                                                                       //
	//Sprawdzanie platynek                                              //
	bLidPuttedCheckEnableShow      						: BOOL;  		//	P030_Recipes.stActRecipe.stUBL.bLidPuttedCheckEnableShow   			// Zezwolenie na prace stacji sprawdzania nakrętek
    lrLidPuttedCheckHeightSVShow 	 					: LREAL;        //    P030_Recipes.stActRecipe.stUBL.lrLidPuttedCheckHeightSVShow			
	lrLidPuttedCheckPositionShow						: LREAL;		//	P030_Recipes.stActRecipe.stUBL.lrLidPuttedCheckPositionShow			// Pozycka sprawdzania platynki
	lrLidPuttedCheckAreaShow							: LREAL;		//	P030_Recipes.stActRecipe.stUBL.lrLidPuttedCheckAreaShow				// [-50...50]  lrLidPuttedCheckPosition +- lrLidPuttedCheckArea. Granica monitorowania 
	iLidPuttedCheckProgramShow							: INT;			//	P030_Recipes.stActRecipe.stUBL.iLidPuttedCheckProgramShow				// Program czujnika wizyjnego 0-20
                                                                        //
	//Zgrzewanie                                                        //
	bLidSealerEnableShow								: BOOL;			//	P030_Recipes.stActRecipe.stUBL.bLidSealerEnableShow				// Zezwolenie na pracę podajnika 
    bLidSealerHeaterEnableShow							: BOOL;			//	P030_Recipes.stActRecipe.stUBL.bLidSealerHeaterEnableShow			// Zezwolenie na prace grzałki  
    iLidSealerHeatingTimeShow							: INT;			//	P030_Recipes.stActRecipe.stUBL.iLidSealerHeatingTimeShow			// Czas zgrzewania  [ms]
	lrLidSealerPressureShow								: LREAL;		//	P030_Recipes.stActRecipe.stUBL.lrLidSealerPressureShow				//	Siła zgrzewania [kg] 
  	lrLidSealerHeightPosSVShow							: LREAL;		//	P030_Recipes.stActRecipe.stUBL.lrLidSealerHeightPosSVShow			// Wysokoć na której ma znajdować się grzałka
	iLidSealerTempHisteresisShow						: INT;			//	P030_Recipes.stActRecipe.stUBL.iLidSealerTempHisteresisShow		// Histereza poprawnej temperatury grzałki (+/- *C), po jej przekroczeniu grzałka wpada w błšd
   	iLidSealer1TempSVShow								: INT;			//	P030_Recipes.stActRecipe.stUBL.iLidSealer1TempSVShow				// Temperatura zadana grzałki 1                                                               
  	iLidSealer2TempSVShow								: INT;			//	P030_Recipes.stActRecipe.stUBL.iLidSealer2TempSVShow				// Temperatura zadana grzałki 2
                                                                        //
	//Przeciąganie zgrzewania                                           //
	bLidSealerDragingStationEnableShow					: BOOL;			//	P030_Recipes.stActRecipe.stUBL.bLidSealerDragingStationEnableShow					// Aktywacja przeciagania formatek pod zakrecarkami
	lrLidSealerDragingStationVelocityShow				: LREAL; 		//	P030_Recipes.stActRecipe.stUBL.lrLidSealerDragingStationVelocityShow				// Prędkosć przeciągania formatek pod zakręcarkami [0-100 %]
    lrLidSealerDragingStationAccelerationShow			: LREAL; 		//	P030_Recipes.stActRecipe.stUBL.lrLidSealerDragingStationAccelerationShow		// Przyspieszenie przeciągania formatek pod podajnikem płatynek 	
    lrLidSealerDragingStationDecelerationShow			: LREAL; 		//	P030_Recipes.stActRecipe.stUBL.lrLidSealerDragingStationDecelerationShow		// Zmniejszenie prędkości przeciągania formatek pod podajnikem płatynek 	
                                                                        //
	//Szlaban podawania zamknięć                            			//	
	bCapFeederGateEnableShow							:BOOL;			//	P030_Recipes.stActRecipe.stUBL.bCapFeederGateEnableShow				// Aktywacja 
	iCapFeederGateBlockingTimeShow						:INT;			//	P030_Recipes.stActRecipe.stUBL.iCapFeederGateBlockingTimeShow		// Czas blokowania
                                                                        //
	//[H] Podajnik zamknięć                        				        //
	bCapFeederEnableShow								:BOOL;			//	P030_Recipes.stActRecipe.stUBL.bCapFeederEnableShow							// [H] Aktywacja
    lrCapFeederHeightPosSVShow							:LREAL:=140;	//	P030_Recipes.stActRecipe.stUBL.lrCapFeederHeightPosSVShow						// [H] Pozycja
	iCapFeederTimeDelayOnShow							:INT; 			//	P030_Recipes.stActRecipe.stUBL.iCapFeederTimeDelayOnShow						// [H] Opóźnienie włączenia
	iCapFeederTimeDelayOffShow							:INT; 			//	P030_Recipes.stActRecipe.stUBL.iCapFeederTimeDelayOffShow						// [H] Opóźnienie wyłączenia
	iCapFeederTimeToEmptySleeveErrorShow				:INT;			//	P030_Recipes.stActRecipe.stUBL.iCapFeederTimeToEmptySleeveErrorShow			// [H] Czas do alarmu pustego rękawa [s] (10-120 s)
                                                                        //
	//Sorter nasadek                                                    //
	//Zmienne z innego sterownika                                       //
	bCapSorterOnlyWeightOKEnableShow					:BOOL;			//	P030_Recipes.stActRecipe.stUBL.bCapSorterOnlyWeightOKEnableShow		// Nakładanie zamknięć tylko na opakowania z waga OK
	                                                                    //
	//Przeciąganie pod sorterem nasadek                                 //
	bCapSorterDragEnableShow							:BOOL;			//	P030_Recipes.stActRecipe.stUBL.bCapSorterDragEnableShow				// [H] Aktywacja
	lrCapSorterDragVelocityShow							:LREAL; 		//	P030_Recipes.stActRecipe.stUBL.lrCapSorterDragVelocityShow				// Prędkość
 	lrCapSorterDragAccelerationShow						:LREAL;			//	P030_Recipes.stActRecipe.stUBL.lrCapSorterDragAccelerationShow			// Przyspieszenie 
	lrCapSorterDragDecelerationShow						:LREAL;			//	P030_Recipes.stActRecipe.stUBL.lrCapSorterDragDecelerationShow			// Hamowanie
                                 				                        //
	//Sprawdzanie nasadki                                      			//	
	bCapPuttedCheckEnableShow							:BOOL;			//	P030_Recipes.stActRecipe.stUBL.bCapPuttedCheckEnableShow				// Aktywacja
    lrCapPuttedCheckHeightPosSVShow						:LREAL:=69;		//	P030_Recipes.stActRecipe.stUBL.lrCapPuttedCheckHeightPosSVShow			// Pozycja
                                 					                    //
	//Zakrecarka szczekowa (Zachować kolejność i opisy!)                //
	bGripperScrewer1EnableShow							:BOOL;			//	P030_Recipes.stActRecipe.stUBL.bGripperScrewer1EnableShow								// Aktywacja 1
	lrGripperScrewingTightTorqueShow					:LREAL;  		//	P030_Recipes.stActRecipe.stUBL.lrGripperScrewingTightTorqueShow						// Nastawa momentu zakręcania [Nm]
	bGripperScrewer2EnableShow							:BOOL;			//	P030_Recipes.stActRecipe.stUBL.bGripperScrewer2EnableShow								// Aktywacja 2
	lrGripperScrewing2TightTorqueShow					:LREAL;  		//	P030_Recipes.stActRecipe.stUBL.lrGripperScrewing2TightTorqueShow						// Nastawa momentu zakręcania 2 [Nm]
	iGripperScrewer1ToolShow							:INT;			//	P030_Recipes.stActRecipe.stUBL.iGripperScrewer1ToolShow								// Wybór narzędzia (1-5), opisy w tablicy AsGripperScrewerTool	
 	lrGripperScrewer1VelocityShow						:LREAL:=6000; 	//	P030_Recipes.stActRecipe.stUBL.lrGripperScrewer1VelocityShow							// Prędkość zakręcania [rpm]
	nGripperScrewer1TightTimeShow						:INT:=100;  	//	P030_Recipes.stActRecipe.stUBL.nGripperScrewer1TightTimeShow							// Czas przytrzymania podczas dokręcania [ms] 	
	iGripperScrewer1StartDelayShow						:INT;			//	P030_Recipes.stActRecipe.stUBL.iGripperScrewer1StartDelayShow							// Zwoka przed zakręcaniem			
	lrGripperScrewerReadyPositionShow					:LREAL := 250;  //	P030_Recipes.stActRecipe.stUBL.lrGripperScrewerReadyPositionShow						// Pozycja gotowości
	lrGripperScrewerPushingCapPositionShow				:LREAL := 250;  //	P030_Recipes.stActRecipe.stUBL.lrGripperScrewerPushingCapPositionShow					// Pozycja docisku  
    lrGripperScrewerScrewingCapPositionShow				:LREAL := 250;  //	P030_Recipes.stActRecipe.stUBL.lrGripperScrewerScrewingCapPositionShow					// Pozycja zakręcania	
    lrGripperScrewerFindScrewPositionShow				:LREAL := 250;  //	P030_Recipes.stActRecipe.stUBL.lrGripperScrewerScrewingCapPositionShow					// Pozycja zakręcania	
	lrGripperScrewerPressureShow						:LREAL;			//	P030_Recipes.stActRecipe.stUBL.lrGripperScrewerPressureShow							// Siła chwytaka nasadki (0.0 kg)
	lrGripperScrewerCatchPressureShow 					:LREAL;			//	P030_Recipes.stActRecipe.stUBL.lrGripperScrewerCatchPressureShow 						// Siła chwytaka butelki (0.0 kg)
	lrDispencerCatchPressureShow 						:LREAL;			//	P030_Recipes.stActRecipe.stUBL.lrDispencerCatchPressureShow 							// Siła chwytaka butelki pod dozownikami (0.0 kg)
	lrGripperScrewerPressureExhaustLevelShow			:LREAL;			//	P030_Recipes.stActRecipe.stUBL.lrGripperScrewerPressureExhaustLevelShow				// Prędkość zamykania chwytaka nasadki (0.0-100.0 %)
	lrGripperScrewerCatchPressureExhaustLevelShow		:LREAL;			//	P030_Recipes.stActRecipe.stUBL.lrGripperScrewerCatchPressureExhaustLevelShow			// Prędkość zamykania chwytaka opakowania (0.0-100.0 %)
	lrGripperScrewerTurnoversToFullScrewedShow			:LREAL;			//	P030_Recipes.stActRecipe.stUBL.lrGripperScrewerTurnoversToFullScrewedShow				// Opakowanie | Ilość obrotów zamknięcia [obr.] (0.5-10.0 obr.)
   	lrGripperScrewerThreadPitchShow						:LREAL;			//	P030_Recipes.stActRecipe.stUBL.lrGripperScrewerThreadPitchShow							// Opakowanie | Skok gwintu [mm] (0.1-10.0 mm)
	lrGripperScrewerThreadTimesShow						:LREAL;			//	P030_Recipes.stActRecipe.stUBL.lrGripperScrewerThreadTimesShow							// Opakowanie | Krotność gwintu [x] (1-10 x)                       		
	nGripperScrewerCatchHeightSVShow					:LREAL:=86;  		//	P030_Recipes.stActRecipe.stUBL.nGripperScrewerCatchHeightSVShow						// Pozycja chwytaka opakowań
	bGripperScrewer1FindScrewShow						:BOOL; 			//	P030_Recipes.stActRecipe.stUBL.bGripperScrewer1FindScrewShow							// Szukanie gwintu w pozycji zakręcania	
	bGripperScrewer1Option4Show							:BOOL;			//	P030_Recipes.stActRecipe.stUBL.bGripperScrewer1Option4Show								// Szukanie gwintu w pozycji dociskania	
	lrGripperScrewer1FindingScrewDegreeShow				:LREAL; 		//	P030_Recipes.stActRecipe.stUBL.lrGripperScrewer1FindingScrewDegreeShow					// Kąt szukania gwintu (max. dla opcji szukania gwintu z czuj. wys.)	
	bGripperScrewer1Option1Show							:BOOL;			//	P030_Recipes.stActRecipe.stUBL.bGripperScrewer1Option1Show								// Otwarty chwytak przy szukaniu gwintu	
	bGripperScrewer1Option2Show							:BOOL;			//	P030_Recipes.stActRecipe.stUBL.bGripperScrewer1Option2Show								// Obrót do tyłu w pozycji dociskania (w trakcie przejazdu do poz. doc.)
	bGripperScrewer1Option3Show							:BOOL;			//	P030_Recipes.stActRecipe.stUBL.bGripperScrewer1Option3Show								// Dodatkowy ruch chwytakiem przed zakręceniem  (w poz. doc.)	
	bGripperScrewer1Option5Show							:BOOL;			//	P030_Recipes.stActRecipe.stUBL.bGripperScrewer1Option5Show								// Szukanie gwintu z czujnikiem wysokości
	bGripperScrewer1Option6Show							:BOOL;			//	P030_Recipes.stActRecipe.stUBL.bGripperScrewer1Option6Show								// Obrót z pozycji docisku do zakręcania
 	bGripperScrewer1Option7Show							:BOOL;			//	P030_Recipes.stActRecipe.stUBL.bGripperScrewer1Option7Show								// Tryb momentowy	
	                                                                    //
	//Przeciaganie formatek pod zakrecarkami                            //
	bBottleDragingStationEnableShow						:BOOL;			//	P030_Recipes.stActRecipe.stUBL.bBottleDragingStationEnableShow				// [H] Aktywacja 
	lrBottleDragingStationVelocityShow					:LREAL; 		//	P030_Recipes.stActRecipe.stUBL.lrBottleDragingStationVelocityShow		// Prędkość
	                                                                    //
	//Sprawdzanie zakręcania                                            //
	bCapCorrectCheckEnableShow							:BOOL;			//	P030_Recipes.stActRecipe.stUBL.bCapCorrectCheckEnableShow					// Aktywacja
    lrCapCorrectCheckHeightPosSVShow					:LREAL:=69;		//	P030_Recipes.stActRecipe.stUBL.lrCapCorrectCheckHeightPosSVShow			// Pozycja
	bCapCorrectCheckCameraEnableShow      				:BOOL;  		//	P030_Recipes.stActRecipe.stUBL.bCapCorrectCheckCameraEnableShow 		// Aktywacja sprawdzania orientacji nasadki
	iCapCorrectCheckCameraProgramShow					:INT;			//	P030_Recipes.stActRecipe.stUBL.iCapCorrectCheckCameraProgramShow		// Program czujnika wizyjnego 0-20
	                                                                    //
	                                                                    //
	//Robot butelek                                                     //
	bBottleTransferEnableShow							:BOOL; 			//	P030_Recipes.stActRecipe.stUBL.bBottleTransferEnableShow					// Aktywacja
	nBottleTransferProgramShow							:UINT; 			//	P030_Recipes.stActRecipe.stUBL.nBottleTransferProgramShow					// [H] Program robota	
	iBottleTransferPickOffsetXShow 						:INT;			//	P030_Recipes.stActRecipe.stUBL.iBottleTransferPickOffsetXShow 				// Offset X pozycji pobrania
	iBottleTransferPickOffsetYShow 						:INT;			//	P030_Recipes.stActRecipe.stUBL.iBottleTransferPickOffsetYShow 				// Offset Y pozycji pobrania  
	iBottleTransferPickOffsetZShow 						:INT; 			//	P030_Recipes.stActRecipe.stUBL.iBottleTransferPickOffsetZShow 				// Offset Z pozycji pobrania
	iBottleTransferPick2OffsetXShow						:INT;			//	P030_Recipes.stActRecipe.stUBL.iBottleTransferPick2OffsetXShow				// Offset X 2 pozycji pobrania
	iBottleTransferPick2OffsetYShow						:INT;  			//	P030_Recipes.stActRecipe.stUBL.iBottleTransferPick2OffsetYShow				// Offset Y 2 pozycji pobrania
	iBottleTransferPick2OffsetZShow						:INT;   		//	P030_Recipes.stActRecipe.stUBL.iBottleTransferPick2OffsetZShow				// Offset Z 2 pozycji pobrania
	iBottleTransferPlace1OffsetXShow 					:INT;			//	P030_Recipes.stActRecipe.stUBL.iBottleTransferPlace1OffsetXShow 			// Offset X pozycji etykieciarki
	iBottleTransferPlace1OffsetYShow 					:INT;  			//	P030_Recipes.stActRecipe.stUBL.iBottleTransferPlace1OffsetYShow 			// Offset Y pozycji etykieciarki
	iBottleTransferPlace1OffsetZShow 					:INT;			//	P030_Recipes.stActRecipe.stUBL.iBottleTransferPlace1OffsetZShow 			// Offset Z pozycji etykieciarki
	iBottleTransferPlace2OffsetXShow 					:INT;			//	P030_Recipes.stActRecipe.stUBL.iBottleTransferPlace2OffsetXShow 			// Offset X pozycji odrzutu
	iBottleTransferPlace2OffsetYShow					:INT;			//	P030_Recipes.stActRecipe.stUBL.iBottleTransferPlace2OffsetYShow			// Offset Y pozycji odrzutu
	iBottleTransferPlace2OffsetZShow 					:INT; 			//	P030_Recipes.stActRecipe.stUBL.iBottleTransferPlace2OffsetZShow 			// Offset Z pozycji odrzutu
	iBottleTransferSpeedShow							:INT := 10;		//	P030_Recipes.stActRecipe.stUBL.iBottleTransferSpeedShow					// Prędkość robota 	
	bBottleTransferInkJetEnableShow						:BOOL;			//	P030_Recipes.stActRecipe.stUBL.bBottleTransferInkJetEnableShow				// Przesuwanie opakowania nad drukarką (Inkjet)
  	bBottleTransferPickOnlyOneShow						:BOOL;			//	P030_Recipes.stActRecipe.stUBL.bBottleTransferPickOnlyOneShow				// [H] Pobieranie tylko 1 opakowania
 	bBottleTransferWeightEnableShow						:BOOL;			//	P030_Recipes.stActRecipe.stUBL.bBottleTransferWeightEnableShow				// Przesuwanie opakowania na wagę 
  	iBottleTransferWeightIntervalShow					:INT;			//	P030_Recipes.stActRecipe.stUBL.iBottleTransferWeightIntervalShow			// Interwał przesuwania na wagę
 	bBottleTransferRotateEnableShow						:BOOL;			//	P030_Recipes.stActRecipe.stUBL.bBottleTransferRotateEnableShow				// Obrót orientacji nasadki   

	//Przeciąganie 
	bBottleTransferAfterDragEnableShow					:BOOL;			// Aktywacja
	                                                                    //
	//Transporter odrzutu                      	                        //
	bBadBottleConveyorEnableShow						:BOOL;			//	P030_Recipes.stActRecipe.stUBL.bBadBottleConveyorEnableShow			// [H] Aktywacja
	nBadBottleConveyorVelocitySVShow					:UINT;			//	P030_Recipes.stActRecipe.stUBL.nBadBottleConveyorVelocitySVShow		// Prędkość
	                                                                    //
	//Etykieciarka                                                      //
	bLabelMachineEnableShow								:BOOL;			//	P030_Recipes.stActRecipe.stUBL.bLabelMachineEnableShow		// Aktywacja
	                                                                    //
	//Stół odbierający                                                  //
	bExitTurnTable1EnableShow							:BOOL;			//	P030_Recipes.stActRecipe.stUBL.bExitTurnTable1EnableShow		// Aktywacja
	//Transporter odbierający                                           //
	bExitConveyorEnableShow								:BOOL;			//	P030_Recipes.stActRecipe.stUBL.bExitConveyorEnableShow				// Aktywacja
	nExitConveyorVelocitySVShow							:UINT;			//	P030_Recipes.stActRecipe.stUBL.nExitConveyorVelocitySVShow			// Prędkość
	                                                                    //
	                                                                    //
	//Transportery główne                                               //
	bFormTransportersEnableShow							:BOOL;			//	P030_Recipes.stActRecipe.stUBL.bFormTransportersEnableShow							// [H] Aktywacja
	nFormTransportersDispencerVelocitySVShow			:UDINT;			//	P030_Recipes.stActRecipe.stUBL.nFormTransportersDispencerVelocitySVShow			// Prędkość transportera przed dozownikami
	nFormTransportersScrewerVelocitySVShow				:UDINT;			//	P030_Recipes.stActRecipe.stUBL.nFormTransportersScrewerVelocitySVShow				// Prędkość transportera za dozownikami
	nFormTransportersAfterCapSorterVelocitySVShow		:UDINT;			//	P030_Recipes.stActRecipe.stUBL.nFormTransportersBeforeScrewerVelocitySVShow		// Prędkość transportera przed zakręcarką
	nFormTransportersBeforeScrewerVelocitySVShow		:UDINT;			//	P030_Recipes.stActRecipe.stUBL.nFormTransportersBeforeScrewerVelocitySVShow		// Prędkość transportera przed zakręcarką
	nFormTransportersSlowerVelocitySVShow				:UDINT;			//	P030_Recipes.stActRecipe.stUBL.nFormTransportersSlowerVelocitySVShow				// Prędkość spowalniacza 
	nFormTransportersAfterScrewerVelocitySVShow			:UDINT;			//	P030_Recipes.stActRecipe.stUBL.nFormTransportersAfterScrewerVelocitySVShow			// Prędkość transportera przed zakręcarką
	nFormTransportersROPPVelocitySVShow					:UDINT;	        //    P030_Recipes.stActRecipe.stUBL.nFormTransportersROPPVelocitySVShow			
	                                                                    //
	//[H] InkJet obwodowy                                               //
	bCircularInkjetEnableShow							:BOOL;			//	P030_Recipes.stActRecipe.stUBL.bCircularInkjetEnableShow			// [H] Aktywacja
	iCircularInkjetSpeedShow							:INT;			//	P030_Recipes.stActRecipe.stUBL.iCircularInkjetSpeedShow			// [H] Prędkość 
	iCircularInkjetDelayShow							:INT;			//	P030_Recipes.stActRecipe.stUBL.iCircularInkjetDelayShow			// [H] Opóźnienie docisku rolek
	iCircularInkjetHoldShow								:INT;			//	P030_Recipes.stActRecipe.stUBL.iCircularInkjetHoldShow				// [H] Czas przytrzymania [ms]
	
	udiCounterExecuteTimeTemp: UDINT;

	//Czujniki Wenglor
	lrMinDistanceToCappedCorrectlyBottleShow			:LREAL; 
	lrMaxDistanceToCappedCorrectlyBottleShow			:LREAL;
	lrSettleTimeMeasuringCappedBottleShow 				:UINT;
	bWenglorSensorCapPuttedShow							:BOOL:=FALSE;
	bWenglorSensorCapCorrectShow						:BOOL:=FALSE;
	bWenglorSensorCapModeShow							:UINT;
	
	//	(***MAIN***)
	//AnRFIDCardNumberShow							:ARRAY [1..100] OF ULINT;	// [H] Tabela numerów formatek 
	//AnRFIDWeightShow								:ARRAY [1..100] OF LREAL;	// [H] Tabela wag formatek	
	
	
END_VAR

VAR_GLOBAL PERSISTENT
	
	(***MAIN***)
	AnRFIDCardNumberShow							:ARRAY [1..100] OF ULINT;	// [H] Tabela numerów formatek 
	AnRFIDWeightShow								:ARRAY [1..100] OF LREAL;	// [H] Tabela wag formatek		

    
	udiCounterGlobal								:UDINT; 					// Globalny licznik [szt.]
	udiCounterGlobalBadBottles						:UDINT;						// Globalny licznik odrzutu [szt.]

	(*****P02_Dispencers****)		
	lrFormsDragingLeftStartPosition					:LREAL;
	lrFormsDragingLeftEndPosition					:LREAL;
	lrFormsDragingRightStartPosition				:LREAL;
	lrFormsDragingRightEndPosition					:LREAL;

	(*****P10_GripperScrewer****)		
	lrBottleDragingStationStartPosition				:LREAL;
	lrBottleDragingStationEndPosition				:LREAL;	
	udiGripperScrewerToolCounter					:UDINT; 	// Licznik kasowalny dla 

	(*****P07_ROPP****)		
	lrROPPDragStationStartPosition					:LREAL;
	lrROPPDragStationEndPosition					:LREAL;	
	
	(*****P08_CapSorter****)		
	lrCapSorterDragStationStartPosition				:LREAL;
	lrCapSorterDragStationEndPosition				:LREAL;	
		
		
	(*****P10_LidSealer****)		
	lrFeedingDragingStationStartPosition				:LREAL;
	lrFeedingDragingStationEndPosition					:LREAL;	
	lrSealingDragingStationStartPosition				:LREAL;
	lrSealingDragingStationEndPosition					:LREAL;		
	
	lrWickFeedingDragingStationStartPosition				:LREAL;
	lrWickFeedingDragingStationEndPosition					:LREAL;	
	
END_VAR

(* stored: Version 1.1.0.1, ProductVersion 3.1.4026.13, FileIdentifier dd0c1903b64182c80646e9069dd7090d385d72d8, FileSignature 23436682d85d42fbd3eb31cb81568c88dc23ea6a311e4698dc5b4bcf0b7407c5297c781630306890e5ca476774dfeead9470573ec0c6fc8b8927748146018f8caa4a42573fc0eafbf4481313686f3e3b2804d03ded93cbe78ae7eab9babc877f7126275d94ddf1cb1631e315cea2a9f684953beef197ae22da272844d3da0c31474dc8486fcd60138d1df5cf85641e51f1415d1c30200de8c71e1361ef4a8a2e6ce5fbc631d1c00069fb0924f50fed62befab576e064f58637feaf9f36d63258dfa4325361bbd331e334669ed5db756a7287effc22ce0d967d6cc979cad62ee64b7c31c5d83e647ebb8e64e29c1f6f61e1f95a0bb41d3ce17bc946b2fdc5ef8e
   GVL VIS: Id {fb1e88ce-5107-422d-b75b-d16f83915954} *)
